KUKA KRL data list: chk_w8_tools_ok.dat

&ACCESS RVO4
&COMMENT Checagem das ferramentas nos docks
DEFDAT chk_w8_tools_ok PUBLIC
ENDDAT
